TYPE ST_ControlElement_HMI_Link EXTENDS ST_BaseControlElement_HMI_Link :
STRUCT
	stControlElement			: ST_ControlElement_HMI;
END_STRUCT
END_TYPE

(* stored: Version 1.1.0.1, ProductVersion 3.1.4024.15
   DUT ST_ControlElement_HMI_Link: Id {638edb7f-1be4-49d0-b6e7-dd9a320886ec} *)
